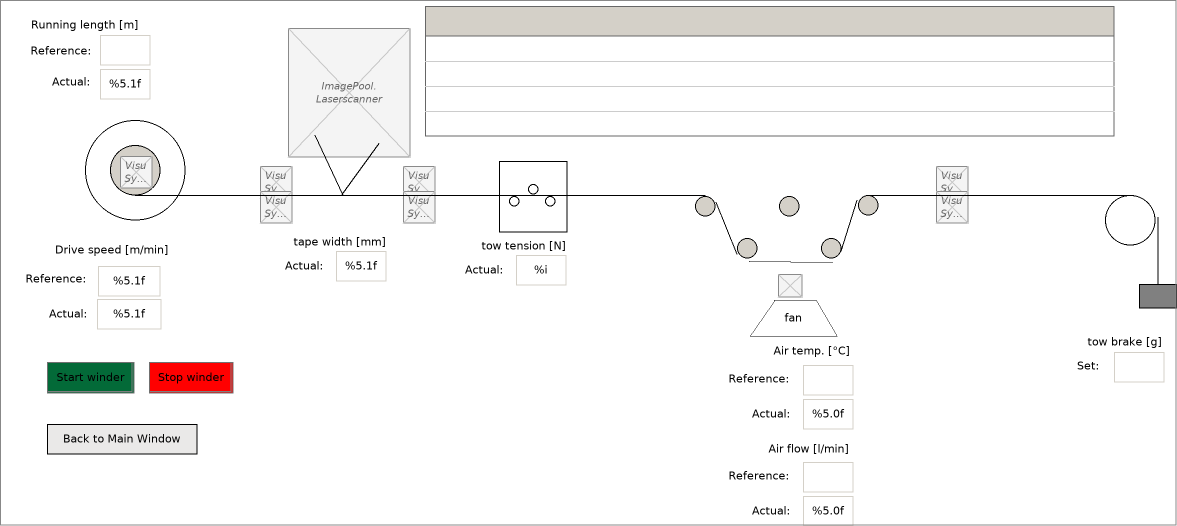
VISUALIZATION Production_Mode  // 1177x526
    Label (10,10 150x30), "Running length [m]"
    Textfield (100,35 50x30)
    Label (37,235 150x30), "Drive speed [m/min]"
    Textfield (97,299 64x30), "%5.1f", text variable: GVL_HMI.ActTapeSpeed
        OnMouseClick: write the text variable via Default
    Label (14,36 80x30), "Reference:"
    Label (13,67 80x30), "Actual:"
    Ellipse (85,120 100x100)
    Ellipse (110,145 50x50)
    Label (10,299 80x30), "Actual:"
    Label (9,264 80x30), "Reference:"
    Image (260,166 32x32), image: VisuSymbols.Symbols.TriangleDown
    Image (260,191 32x32), image: VisuSymbols.Symbols.TriangleUp
    Image (403,166 32x32), image: VisuSymbols.Symbols.TriangleDown
    Image (403,191 32x32), image: VisuSymbols.Symbols.TriangleUp
    Ellipse (695,196 20x20)
    Ellipse (737,238 20x20)
    Ellipse (779,196 20x20)
    Ellipse (821,238 20x20)
    Ellipse (858,195 20x20)
    Image (936,166 32x32), image: VisuSymbols.Symbols.TriangleDown
    Image (936,191 32x32), image: VisuSymbols.Symbols.TriangleUp
    Label (753,336 100x30), "Air temp. [°C]"
    Textfield (803,399 50x30), "%5.0f", text variable: GVL_Axis.rWinderVelocity
        OnMouseClick: write the text variable via Default
    Textfield (803,365 50x30)
    Label (713,399 80x30), "Actual:"
    Label (712,364 80x30), "Reference:"
    Label (752,434 100x30), "Air flow [l/min]"
    Textfield (803,496 50x30), "%5.0f", text variable: GVL_Axis.rWinderVelocity
        OnMouseClick: write the text variable via Default
    Textfield (803,462 50x30)
    Label (713,496 80x30), "Actual:"
    Label (712,461 80x30), "Reference:"
    Label (275,227 114x30), "tape width [mm]"
    Textfield (336,251 50x30), "%5.1f", text variable: GVL_Axis.rWinderVelocity
        OnMouseClick: write the text variable via Default
    Label (246,251 80x30), "Actual:"
    Polygon (775,300) (774,300) (816,300) (837,336) (750,336), "fan"
    Image (778,274 24x23), image: VisuSymbols.Symbols.ArrowBoldUp
    Line (737,254) (716,202)
    Line (749,261) (832,262)
    Label (455,231 114x30), "tow tension [N]"
    Textfield (516,255 50x30), "%i", text variable: GVL.iTensionMonitoringData
        OnMouseClick: write the text variable via Default
    Label (426,255 80x30), "Actual:"
    Label (1051,327 114x30), "tow brake [g]"
    Label (1022,351 80x30), "Set:"
    Textfield (1114,352 50x30)
    Table (425,6 689x130), data array: GVL.LaserScannerData
        p3854506369: GVL.LaserScannerData[INDEX]
    Rectangle (47,424 150x30), "Back to Main Window"
        OnMouseClick: change screen: MainWindow
    Textfield (100,69 50x30), "%5.1f", text variable: GVL_HMI.RunningLength
        OnMouseClick: write the text variable via Default
    Rectangle (499,161 68x71)
    Ellipse (509,196 10x10)
    Ellipse (528,184 10x10)
    Ellipse (545,196 10x10)
    Line (135,195) (705,195)
    Line (841,251) (857,200)
    Line (867,195) (1132,195)
    Ellipse (1105,195 50x50)
    Line (1158,288) (1158,217)
    Rectangle (1139,284 38x24)
    Image (288,28 122x129), image: ImagePool.Laserscanner
    Line (342,194) (379,143)
    Line (343,195) (315,135)
    Textfield (98,266 62x30), "%5.1f", text variable: GVL_Axis.rWinderVelocity
        OnMouseClick: write the text variable via VisuDialogs.Numpad, min 2.7, max 15
    Button (47,362 87x31), "Start winder", colour toggle: GVL_HMI.bButtonStartWinder
        OnMouseDown: execute { GVL_HMI.bButtonStartWinder := TRUE; }
        OnMouseUp: execute { GVL_HMI.bButtonStartWinder := FALSE; }
    Button (149,362 84x31), "Stop winder", colour toggle: GVL_HMI.bButtonStopWinder
        OnMouseDown: execute { GVL_HMI.bButtonStopWinder := TRUE; }
        OnMouseUp: execute { GVL_HMI.bButtonStopWinder := FALSE; }
    Image (120,156 32x32), image: VisuSymbols.Symbols.ArrowHalfRightUp
END_VISUALIZATION

(* stored: Version 1.1.0.1
   Visu Production_Mode: Id {54e80f91-dfb9-4954-9114-9332cd794b3e} *)
